// TwinCAT 3 PLC project SimpleEventMessage
// ProgramVersion: 3.1.4023.0
// libraries:
//   Tc2_Standard, * (Beckhoff Automation GmbH)
//   Tc2_System, * (Beckhoff Automation GmbH)
//   Tc3_EventLogger, * (Beckhoff Automation GmbH)
//   Tc3_Module, * (Beckhoff Automation GmbH)
// project tree:
//   EventLoggerClass/ ITcMessage_Ext.TcIO, TcMessage_Ext.TcPOU (not stored)
//   / PlcTask.TcTTO
//   POUs/ MAIN.TcPOU
// real-time tasks:
//   TASK PlcTask: cycle T#10ms, priority 20, ADS port 350

CONFIGURATION SimpleEventMessage
    RESOURCE PLC ON TwinCAT3
        TASK PlcTask(INTERVAL := T#10ms, PRIORITY := 20);
        PROGRAM MAIN WITH PlcTask : MAIN;
    END_RESOURCE
END_CONFIGURATION

// ---- EventLoggerClass/ITcMessage_Ext.TcIO
INTERFACE ITcMessage_Ext

PROPERTY LoggerLevel : TcEventSeverity
GET
END_GET
SET
END_SET
END_PROPERTY

METHOD Send : BOOL
VAR_INPUT
	eventType : Tc3_EventLogger.TcEventEntry;
	args : STRING(255);
END_VAR
END_METHOD

END_INTERFACE

// ---- POUs/MAIN.TcPOU
PROGRAM MAIN
VAR
	Logger : TcMessage_Ext := (LoggerLevel := TcEventSeverity.Verbose);
	iLogger : ITcMessage_Ext := Logger;
	bSendHello : BOOL;
	bSendError : BOOL;
END_VAR

IF bSendHello THEN
	iLogger.Send(Tc_Events.TestEventClass.Hello,' Bob');
	bSendHello := FALSE;	
END_IF

IF bSendError THEN
	iLogger.Send(Tc_Events.TestEventClass.Error, 'Oh dear');
	bSendError := FALSE;
END_IF

END_PROGRAM
